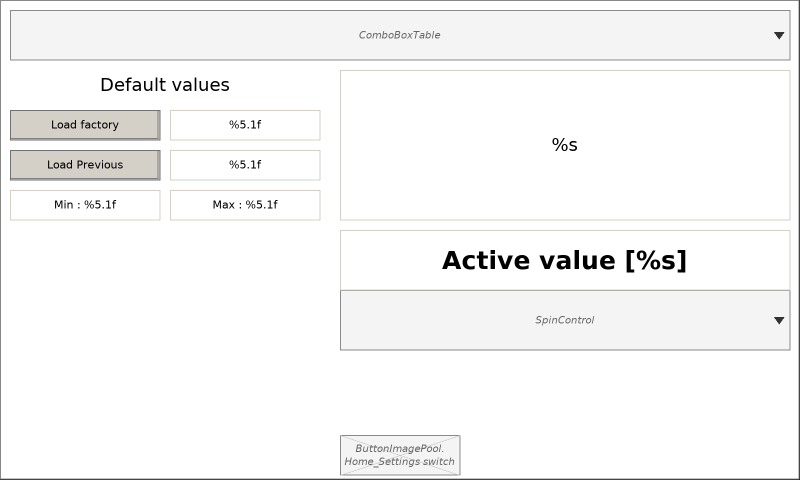
VISUALIZATION ParameterScreen  // 800x480
    Rectangle (0,0 800x480)
    ComboBoxTable (10,10 780x50), variable: GVL_Parameters.fbParameterHandler.nLookupIndex, data array: GVL_Parameters.fbParameterHandler.arParameters
        p1128707560: GVL_Parameters.fbParameterHandler.nNumberOfParameters
        p3854506369: GVL_Parameters.fbParameterHandler.arParameters[INDEX].nNumber
        p1892666644: GVL_Parameters.fbParameterHandler.arParameters[INDEX].sName
        p338671338: GVL_Parameters.fbParameterHandler.arParameters[INDEX].sType
        p2170511999: GVL_Parameters.fbParameterHandler.arParameters[INDEX].pParameter^
    Group (10,70 310x150)
        Button (0,40 150x30), "Load factory"
            tap GVL_Parameters.fbParameterHandler.bCmdLoadfactory
        Label (0,0 310x30), "Default values"
        Textfield (160,40 150x30), "%5.1f", text variable: GVL_Parameters.fbParameterHandler.arParameters[GVL_Parameters.fbParameterHandler.nLookupIndex].pParameter^.fFactory
            OnMouseClick: write the text variable via VisuDialogs.Numpad, min GVL_Parameters.fbParameterHandler.arParameters[GVL_Parameters.fbParameterHandler.nLookupIndex].pParameter^.fMinimum, max GVL_Parameters.fbParameterHandler.arParameters[GVL_Parameters.fbParameterHandler.nLookupIndex].pParameter^.fMaximum
        Button (0,80 150x30), "Load Previous"
            tap GVL_Parameters.fbParameterHandler.bCmdLoadFromPrevious
        Textfield (160,80 150x30), "%5.1f", text variable: GVL_Parameters.fbParameterHandler.arParameters[GVL_Parameters.fbParameterHandler.nLookupIndex].pParameter^.fSaved
        Textfield (160,120 150x30), "Max : %5.1f", text variable: GVL_Parameters.fbParameterHandler.arParameters[GVL_Parameters.fbParameterHandler.nLookupIndex].pParameter^.fMaximum
            OnMouseClick: write the text variable via VisuDialogs.Numpad
        Textfield (0,120 150x30), "Min : %5.1f", text variable: GVL_Parameters.fbParameterHandler.arParameters[GVL_Parameters.fbParameterHandler.nLookupIndex].pParameter^.fMinimum
            OnMouseClick: write the text variable via VisuDialogs.Numpad
    Textfield (340,70 450x150), "%s", text variable: GVL_Parameters.fbParameterHandler.arParameters[GVL_Parameters.fbParameterHandler.nLookupIndex].pParameter^.sDiscription
    SpinControl (340,290 450x60), variable: GVL_Parameters.fbParameterHandler.arParameters[GVL_Parameters.fbParameterHandler.nLookupIndex].pParameter^.fValue
        p576042468: GVL_Parameters.fbParameterHandler.arParameters[GVL_Parameters.fbParameterHandler.nLookupIndex].pParameter^.fMinimum
        p651134158: GVL_Parameters.fbParameterHandler.arParameters[GVL_Parameters.fbParameterHandler.nLookupIndex].pParameter^.fMaximum
        OnMouseClick: write the text variable via VisuDialogs.Numpad, min GVL_Parameters.fbParameterHandler.arParameters[GVL_Parameters.fbParameterHandler.nLookupIndex].pParameter^.fMinimum, max GVL_Parameters.fbParameterHandler.arParameters[GVL_Parameters.fbParameterHandler.nLookupIndex].pParameter^.fMaximum
    Textfield (340,230 450x60), "Active value [%s]", text variable: GVL_Parameters.fbParameterHandler.arParameters[GVL_Parameters.fbParameterHandler.nLookupIndex].pParameter^.sUnit
    Image (340,435 120x40), image: ButtonImagePool.Home_Settings switch
        OnMouseClick: execute { GVL_HMI.nStartVisu := E_StartVisu.Logo ; }
        OnMouseClick: toggle GVL_Parameters.fbParameterHandler.bCmdParFileWrite
END_VISUALIZATION

(* stored: Version 1.1.0.1, ProductVersion 3.1.4024.5
   Visu ParameterScreen: Id {be090142-cc46-445b-bfe3-261de64e9afe} *)
